FUNCTION_BLOCK F_INT_TO_USINT (* convert INT to USINT *)
  (* Standard: 61131-3; Classification: type conversion function *)
  (* Version 0.0, 2011-12-25, 4DIAC-IDE, 4DIAC-Consortium *)
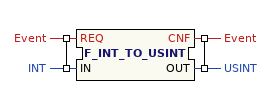
  EVENT_INPUT
    REQ WITH IN; (* Service Request *)
  END_EVENT
  EVENT_OUTPUT
    CNF WITH OUT; (* Confirmation of Requested Service *)
  END_EVENT
  VAR_INPUT
    IN : INT; (* Input Value *)
  END_VAR
  VAR_OUTPUT
    OUT : USINT; (* Output Value *)
  END_VAR
  SERVICE APPLICATION/RESOURCE (* convert INT to USINT *)
    SEQUENCE normal_establishment
      APPLICATION.INIT+(PARAMS) -> APPLICATION.INITO+(PARAMS);
    END_SEQUENCE
    SEQUENCE unsuccessful_establishment
      APPLICATION.INIT+(PARAMS) -> APPLICATION.INITO-(STATUS);
    END_SEQUENCE
    SEQUENCE request_confirm
      APPLICATION.REQ+(SD) -> APPLICATION.CNF+(RD);
    END_SEQUENCE
    SEQUENCE request_inhibited
      APPLICATION.REQ-(SD) -> APPLICATION.CNF-(STATUS);
    END_SEQUENCE
    SEQUENCE request_error
      APPLICATION.REQ+(SD) -> APPLICATION.CNF-(STATUS);
    END_SEQUENCE
    SEQUENCE indication_response
      RESOURCE.indicate(RD) -> APPLICATION.IND+(RD);
      APPLICATION.RSP(QI,SD) -> RESOURCE.response(QI,SD);
    END_SEQUENCE
    SEQUENCE indication_inhibited
      RESOURCE.indicate(RD,QI=FALSE) -> RESOURCE.inhibited();
    END_SEQUENCE
    SEQUENCE error_indication
      RESOURCE.error(STATUS) -> APPLICATION.IND-(STATUS);
    END_SEQUENCE
    SEQUENCE application_initiated_termination
      APPLICATION.INIT-() -> APPLICATION.INITO-(STATUS);
    END_SEQUENCE
    SEQUENCE resource_initiated_termination
      -> APPLICATION.INITO-(STATUS);
    END_SEQUENCE
  END_SERVICE
END_FUNCTION_BLOCK
